FUNCTION_BLOCK HandshakeStateMachine (* Template for a simple Basic Function Block Type *)
  (* Standard: 61499-2 *)
  (* Version 1.0, 2019-12-04, Mario *)
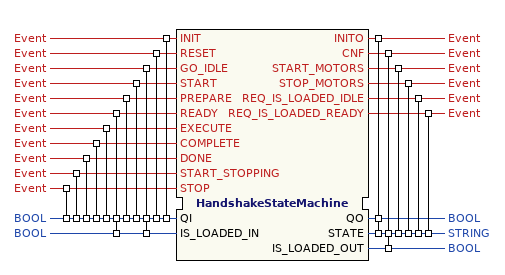
  EVENT_INPUT
    INIT WITH QI; (* Initialization Request *)
    RESET WITH QI; (* Reset Handshake *)
    GO_IDLE WITH IS_LOADED_IN, QI; (* Go to Idle_loaded/Idle_empty depending on QI *)
    START WITH QI; (* Go to Starting State *)
    PREPARE WITH QI; (* Prepare for handshake *)
    READY WITH IS_LOADED_IN, QI; (* Go to readyLoaded/readyEmpty depending on QI *)
    EXECUTE WITH QI; (* Execute handshake *)
    COMPLETE WITH QI; (* Start completing handshake *)
    DONE WITH QI; (* Complete handshake *)
    START_STOPPING WITH QI; (* Prepare to stop *)
    STOP WITH QI; (* Stop *)
  END_EVENT
  EVENT_OUTPUT
    INITO WITH STATE, QO; (* Initialization Confirm *)
    CNF WITH STATE, IS_LOADED_OUT; (* Execution Confirmation *)
    START_MOTORS WITH STATE; (* Starts the motors *)
    STOP_MOTORS WITH STATE; (* Stop all motors *)
    REQ_IS_LOADED_IDLE WITH STATE; (* Request Conveyor Loaded for IDLE? (QI) *)
    REQ_IS_LOADED_READY WITH STATE; (* Request Conveyor Loaded for READY? (QI) *)
  END_EVENT
  VAR_INPUT
    QI : BOOL; (* Should always be 1 *)
    IS_LOADED_IN : BOOL; (* Is the conveyor loaded? *)
  END_VAR
  VAR_OUTPUT
    QO : BOOL;
    STATE : STRING; (* Pass on current state *)
    IS_LOADED_OUT : BOOL;
  END_VAR
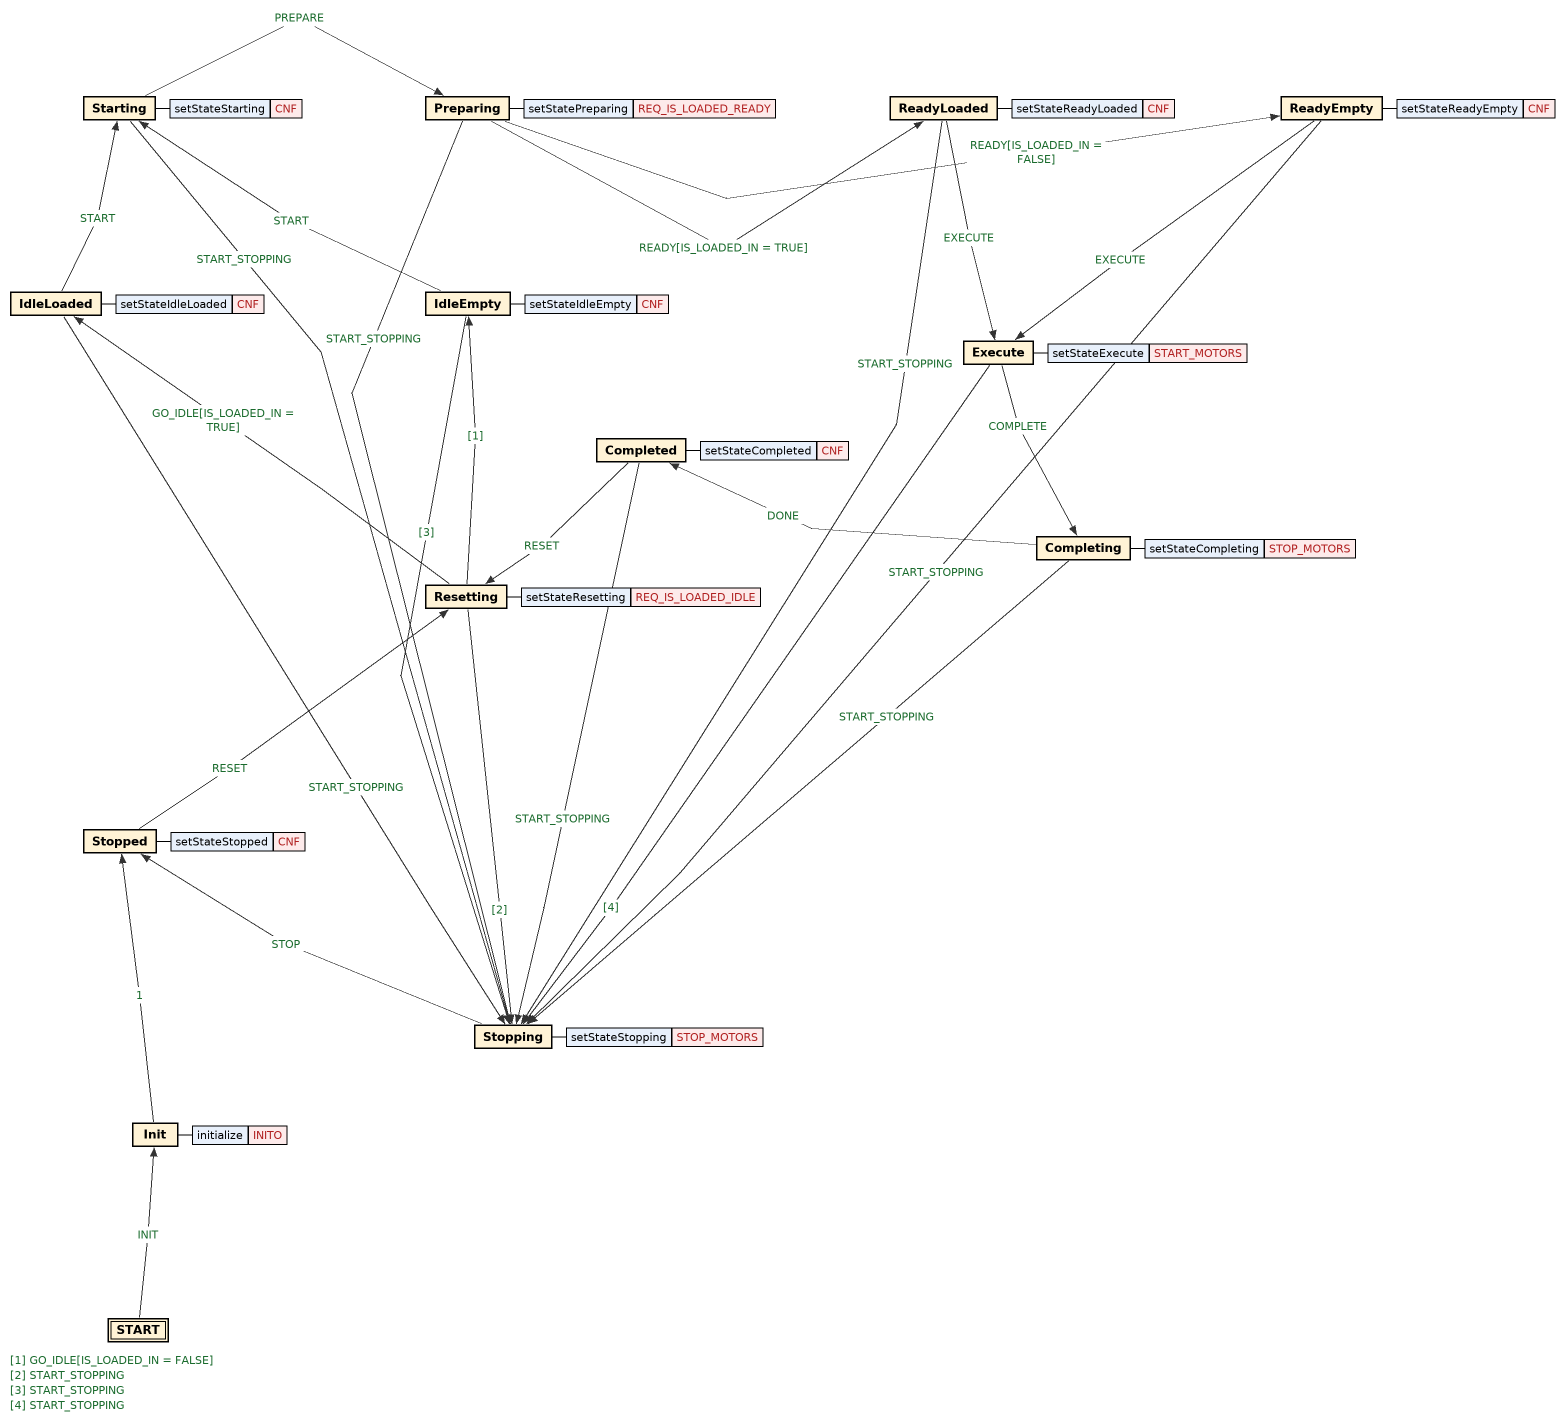
  EC_STATES
    START; (* Initial State *)
    Starting : setStateStarting -> CNF;
    Preparing : setStatePreparing -> REQ_IS_LOADED_READY;
    ReadyLoaded : setStateReadyLoaded -> CNF;
    ReadyEmpty : setStateReadyEmpty -> CNF;
    Execute : setStateExecute -> START_MOTORS;
    Completed : setStateCompleted -> CNF;
    Completing : setStateCompleting -> STOP_MOTORS;
    Resetting : setStateResetting -> REQ_IS_LOADED_IDLE;
    IdleEmpty : setStateIdleEmpty -> CNF;
    IdleLoaded : setStateIdleLoaded -> CNF;
    Stopping : setStateStopping -> STOP_MOTORS;
    Stopped : setStateStopped -> CNF;
    Init : initialize -> INITO;
  END_STATES
  EC_TRANSITIONS
    Stopping TO Stopped := STOP;
    Stopped TO Resetting := RESET;
    Resetting TO IdleEmpty := GO_IDLE[IS_LOADED_IN = FALSE];
    Resetting TO IdleLoaded := GO_IDLE[IS_LOADED_IN = TRUE];
    IdleLoaded TO Starting := START;
    IdleEmpty TO Starting := START;
    Starting TO Preparing := PREPARE;
    Preparing TO ReadyEmpty := READY[IS_LOADED_IN = FALSE];
    Preparing TO ReadyLoaded := READY[IS_LOADED_IN = TRUE];
    ReadyLoaded TO Execute := EXECUTE;
    ReadyEmpty TO Execute := EXECUTE;
    Execute TO Completing := COMPLETE;
    Completing TO Completed := DONE;
    Completed TO Resetting := RESET;
    IdleLoaded TO Stopping := START_STOPPING;
    Resetting TO Stopping := START_STOPPING;
    Completing TO Stopping := START_STOPPING;
    Starting TO Stopping := START_STOPPING;
    IdleEmpty TO Stopping := START_STOPPING;
    Preparing TO Stopping := START_STOPPING;
    ReadyLoaded TO Stopping := START_STOPPING;
    Execute TO Stopping := START_STOPPING;
    ReadyEmpty TO Stopping := START_STOPPING;
    START TO Init := INIT;
    Init TO Stopped := 1;
    Completed TO Stopping := START_STOPPING;
  END_TRANSITIONS
  ALGORITHM initialize IN ST: (* Initialization algorithm *)
QO := QI;
STATE := "NOT INITIALIZED";
  END_ALGORITHM
  ALGORITHM deInitialize IN ST: (* Normally executed algorithm *)
QO := FALSE;
  END_ALGORITHM
  ALGORITHM setStateStopped IN ST: (* new algorithm *)
STATE := "STOPPED";
  END_ALGORITHM
  ALGORITHM setStateStopping IN ST: (* new algorithm *)
STATE :="STOPPING";
  END_ALGORITHM
  ALGORITHM setStateResetting IN ST: (* new algorithm *)
STATE := "RESETTING";
  END_ALGORITHM
  ALGORITHM setStateIdleLoaded IN ST: (* new algorithm *)
STATE := "IDLE_LOADED";
IS_LOADED_OUT := TRUE;
  END_ALGORITHM
  ALGORITHM setStateIdleEmpty IN ST: (* new algorithm *)
STATE := "IDLE_EMPTY";
IS_LOADED_OUT := FALSE;
  END_ALGORITHM
  ALGORITHM setStateStarting IN ST: (* new algorithm *)
STATE := "STARTING";
  END_ALGORITHM
  ALGORITHM setStatePreparing IN ST: (* new algorithm *)
STATE := "PREPARING";
  END_ALGORITHM
  ALGORITHM setStateReadyLoaded IN ST: (* new algorithm *)
STATE := "READY_LOADED";
  END_ALGORITHM
  ALGORITHM setStateReadyEmpty IN ST: (* new algorithm *)
STATE := "READY_EMPTY";
  END_ALGORITHM
  ALGORITHM setStateExecute IN ST: (* new algorithm *)
STATE := "EXECUTE";
  END_ALGORITHM
  ALGORITHM setStateCompleting IN ST: (* new algorithm *)
STATE := "COMPLETING";
  END_ALGORITHM
  ALGORITHM setStateCompleted IN ST: (* new algorithm *)
STATE := "COMPLETE";
  END_ALGORITHM
END_FUNCTION_BLOCK
